SUBAPPLICATION Ventilsteuerung_Uebung_071a (* WBSD auf UT ausgeben, Q1 Schalten wenn Speed &gt;0 *)
  (* Standard: 61499-2 *)
  (* Version 1.0, 2023-10-23, franz *)
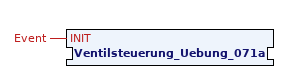
  EVENT_INPUT
    INIT;
  END_EVENT
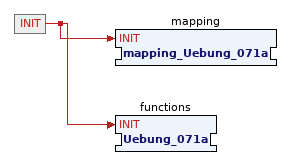
  SUBAPPS
    mapping : mapping_Uebung_071a;
    functions : Uebung_071a;
  END_SUBAPPS
  EVENT_CONNECTIONS
    INIT TO mapping.INIT;
    INIT TO functions.INIT;
  END_CONNECTIONS
END_SUBAPPLICATION
